FUNCTION_BLOCK ServiceExample (* Switching (demultiplexing) an event based on boolean input G *)
  (* Standard: 61499-1 Annex A; Description: Copyright (c) 2017 fortiss GmbH This program and the accompanying materials are made available under the terms of the Eclipse Public License 2.0 which is available at https://www.eclipse.org/legal/epl-2.0/ SPDX-License-Identifier: EPL-2.0 *)
  (* Version 1.0, 2017-09-21, Alois Zoitl, fortiss GmbH, initial API and implementation and/or initial documentation *)
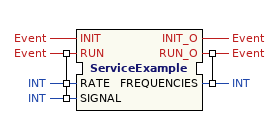
  EVENT_INPUT
    INIT;
    RUN WITH RATE, SIGNAL;
  END_EVENT
  EVENT_OUTPUT
    INIT_O;
    RUN_O WITH FREQUENCIES;
  END_EVENT
  VAR_INPUT
    RATE : INT; {SET_ATTRIBUTE(OpcUa, Constant)}
    SIGNAL : INT; {SET_ATTRIBUTE(OpcUa, Variable)}
  END_VAR
  VAR_OUTPUT
    FREQUENCIES : INT; {SET_ATTRIBUTE(OpcUa, Variable)}
  END_VAR
END_FUNCTION_BLOCK
(* other elements stored in the file *)
(* SelfDiscription FBType=SERVICE *)
